// TIA Portal V20 export
DATA_BLOCK "BK07"   // DB233
// stored: MemoryReserve 100
   VAR
      "X10-1 TAPE ATTACHMENT VACUUM PRESSURE SWITCH" : Bool;
      "X10-2 SPARE" : Bool;
      "X12-1 TOP TAPE ATTACHMENT UP" : Bool;
      "X12-2 TOP TAPE ATTACHMENT DOWN" : Bool;
      "X14-1 TOP TAPING X-AXIS LIMIT SENSOR(-)" : Bool;
      "X14-2 TOP TAPING X-AXIS HOMING SENSOR" : Bool;
      "X16-1 TOP TAPING X-AXIS LIMIT SENSOR(+)" : Bool;
      "X16-2 SPARE" : Bool;
   END_VAR
BEGIN
END_DATA_BLOCK
